% RSLogix 500 project proj_finale_BAK014.RSS, saved by version 8.30.00.16 %
PROJECT "UNTITLED"    % processor: MicroLogix 1000 %

PROGRAM FILES
  LAD 2 "MAIN_PROG"  5 rungs
  LAD 3 "USER_FAULT"  1 rungs
  LAD 4 "HSC_INT"  1 rungs
  LAD 5 "STI_INT"  1 rungs
  LAD 6, 7, 8, 9, 10, 11, 12, 13, 14, 15, 16: only END

DATA FILES
  O0 OUTPUT  1 elements
  I1 INPUT  2 elements
  S2 STATUS  33 elements
  B3 BINARY  32 elements
  T4 TIMER  40 elements
  C5 COUNTER  32 elements
  R6 CONTROL  16 elements
  N7 INTEGER  105 elements

LADDER 2 "MAIN_PROG"
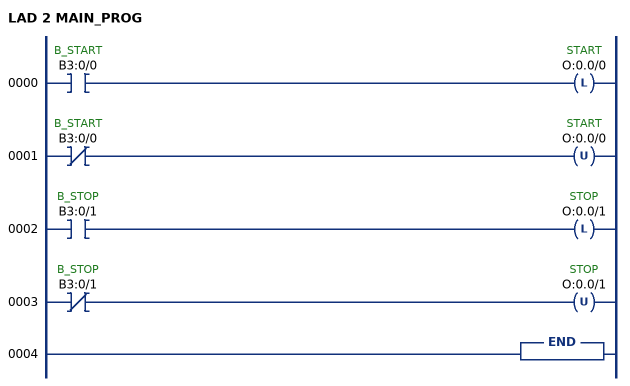
% Rung: 0 %
SOR XIC B3:0/0 OTL O:0.0/0 EOR
%   B3:0/0  B_START %
%   O:0.0/0  START %
% Rung: 1 %
SOR XIO B3:0/0 OTU O:0.0/0 EOR
%   B3:0/0  B_START %
%   O:0.0/0  START %
% Rung: 2 %
SOR XIC B3:0/1 OTL O:0.0/1 EOR
%   B3:0/1  B_STOP %
%   O:0.0/1  STOP %
% Rung: 3 %
SOR XIO B3:0/1 OTU O:0.0/1 EOR
%   B3:0/1  B_STOP %
%   O:0.0/1  STOP %
% Rung: 4 %
SOR END EOR

OTHER DOCUMENTED ADDRESSES
  N7:0  VARETAT
  O:0.0/2  CATALYSEUR

DATA TABLE (non-zero values as saved)
DATA B3
% B3:0 % 0X0001 0X0000 0X0000 0X0000 0X0000 0X0000 0X0000 0X0000 0X0000 0X0000
DATA N7
% N7:0 % 1 0 0 0 0 0 0 0 0 0
